// TIA Portal V19 export
TYPE "LEXCHANGETRAY_typeRollerIoSignalControlNode_B2"
// reset: Bool
// monitoring: LEXCHANGETRAY_typeRollerIoSignalContronNodeMonitoring_B2
// stored: Access Published
   STRUCT
      reset : Bool;
      monitoring { S7_SetPoint := 'True'} : "LEXCHANGETRAY_typeRollerIoSignalContronNodeMonitoring_B2";
   END_STRUCT;
END_TYPE
